(* Logix 5000 project; controller BTS01 vendor 1 type 14 code 217 rev 32.14; software revision 32.04; part 9 of 15 *)
(* tags used below, declared in another part *)
   Alarm_Active : DINT;
   Alarm_TMR : TIMER[17,32];
   ALM_ENABLE : DINT[25];
   HMI_Global_Alarm_Ack_PB : BOOL;
   HMIAlarms : DINT[25];   // Alarm Trigger Array
   HMIAlarmsMsg : STRING64[17,32];   // Alarm Descriptions to Match Alarm Trigger Array
(* Alarm, continued *)

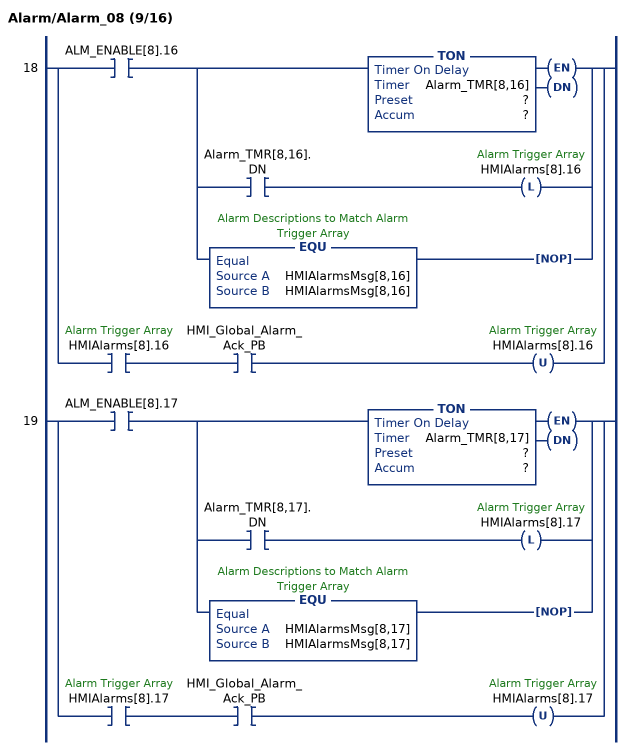
   [picture p159: Alarm/Alarm_08 rungs 18-19]
   18: [XIC(ALM_ENABLE[8].16) [TON(Alarm_TMR[8,16],?,?) ,XIC(Alarm_TMR[8,16].DN) OTL(HMIAlarms[8].16) ,EQU(HMIAlarmsMsg[8,16],HMIAlarmsMsg[8,16]) NOP() ] ,XIC(HMIAlarms[8].16) XIC(HMI_Global_Alarm_Ack_PB) OTU(HMIAlarms[8].16) ];
   19: [XIC(ALM_ENABLE[8].17) [TON(Alarm_TMR[8,17],?,?) ,XIC(Alarm_TMR[8,17].DN) OTL(HMIAlarms[8].17) ,EQU(HMIAlarmsMsg[8,17],HMIAlarmsMsg[8,17]) NOP() ] ,XIC(HMIAlarms[8].17) XIC(HMI_Global_Alarm_Ack_PB) OTU(HMIAlarms[8].17) ];
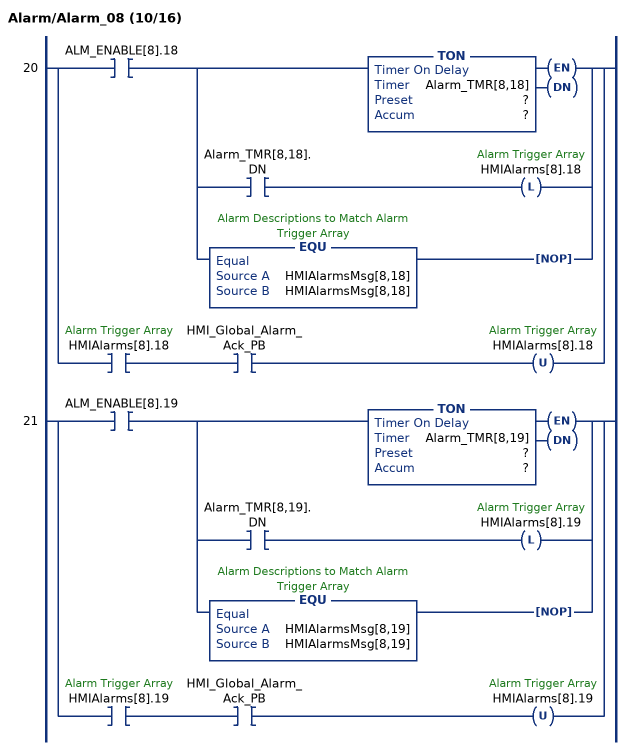
   20: [XIC(ALM_ENABLE[8].18) [TON(Alarm_TMR[8,18],?,?) ,XIC(Alarm_TMR[8,18].DN) OTL(HMIAlarms[8].18) ,EQU(HMIAlarmsMsg[8,18],HMIAlarmsMsg[8,18]) NOP() ] ,XIC(HMIAlarms[8].18) XIC(HMI_Global_Alarm_Ack_PB) OTU(HMIAlarms[8].18) ];
   21: [XIC(ALM_ENABLE[8].19) [TON(Alarm_TMR[8,19],?,?) ,XIC(Alarm_TMR[8,19].DN) OTL(HMIAlarms[8].19) ,EQU(HMIAlarmsMsg[8,19],HMIAlarmsMsg[8,19]) NOP() ] ,XIC(HMIAlarms[8].19) XIC(HMI_Global_Alarm_Ack_PB) OTU(HMIAlarms[8].19) ];
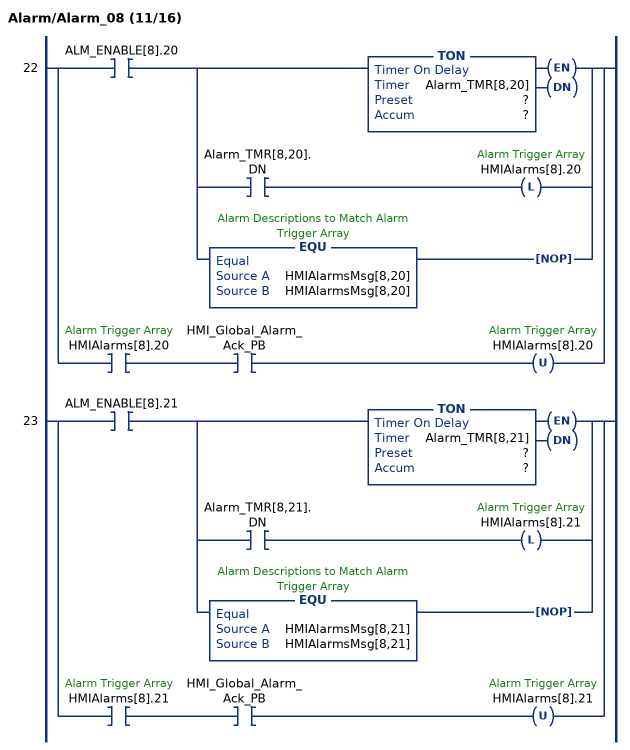
   22: [XIC(ALM_ENABLE[8].20) [TON(Alarm_TMR[8,20],?,?) ,XIC(Alarm_TMR[8,20].DN) OTL(HMIAlarms[8].20) ,EQU(HMIAlarmsMsg[8,20],HMIAlarmsMsg[8,20]) NOP() ] ,XIC(HMIAlarms[8].20) XIC(HMI_Global_Alarm_Ack_PB) OTU(HMIAlarms[8].20) ];
   23: [XIC(ALM_ENABLE[8].21) [TON(Alarm_TMR[8,21],?,?) ,XIC(Alarm_TMR[8,21].DN) OTL(HMIAlarms[8].21) ,EQU(HMIAlarmsMsg[8,21],HMIAlarmsMsg[8,21]) NOP() ] ,XIC(HMIAlarms[8].21) XIC(HMI_Global_Alarm_Ack_PB) OTU(HMIAlarms[8].21) ];
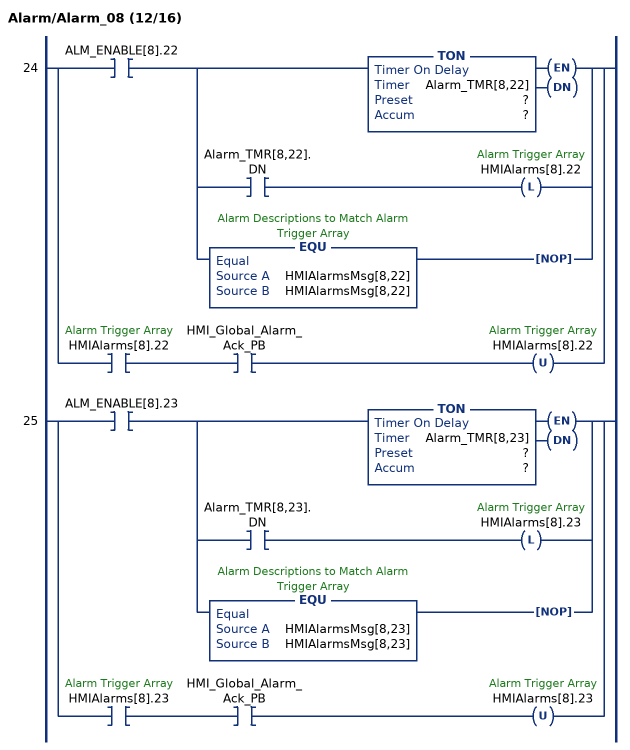
   24: [XIC(ALM_ENABLE[8].22) [TON(Alarm_TMR[8,22],?,?) ,XIC(Alarm_TMR[8,22].DN) OTL(HMIAlarms[8].22) ,EQU(HMIAlarmsMsg[8,22],HMIAlarmsMsg[8,22]) NOP() ] ,XIC(HMIAlarms[8].22) XIC(HMI_Global_Alarm_Ack_PB) OTU(HMIAlarms[8].22) ];
   25: [XIC(ALM_ENABLE[8].23) [TON(Alarm_TMR[8,23],?,?) ,XIC(Alarm_TMR[8,23].DN) OTL(HMIAlarms[8].23) ,EQU(HMIAlarmsMsg[8,23],HMIAlarmsMsg[8,23]) NOP() ] ,XIC(HMIAlarms[8].23) XIC(HMI_Global_Alarm_Ack_PB) OTU(HMIAlarms[8].23) ];
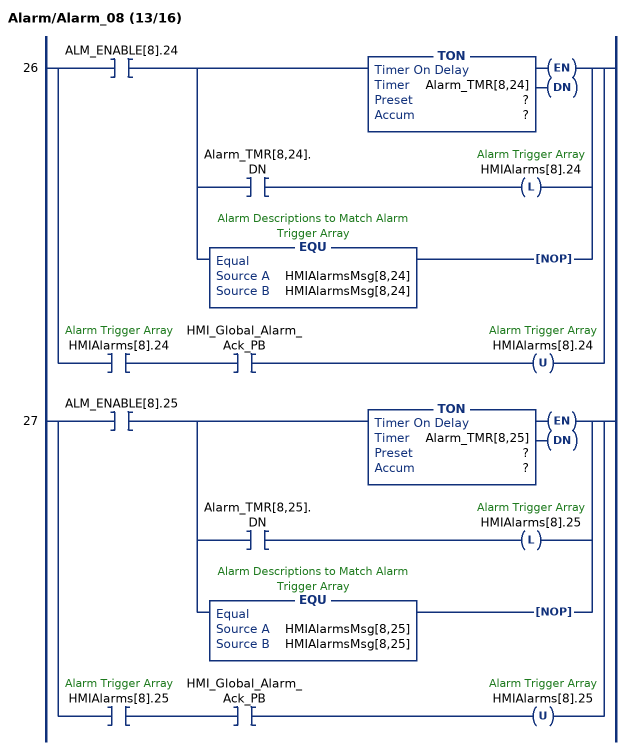
   26: [XIC(ALM_ENABLE[8].24) [TON(Alarm_TMR[8,24],?,?) ,XIC(Alarm_TMR[8,24].DN) OTL(HMIAlarms[8].24) ,EQU(HMIAlarmsMsg[8,24],HMIAlarmsMsg[8,24]) NOP() ] ,XIC(HMIAlarms[8].24) XIC(HMI_Global_Alarm_Ack_PB) OTU(HMIAlarms[8].24) ];
   27: [XIC(ALM_ENABLE[8].25) [TON(Alarm_TMR[8,25],?,?) ,XIC(Alarm_TMR[8,25].DN) OTL(HMIAlarms[8].25) ,EQU(HMIAlarmsMsg[8,25],HMIAlarmsMsg[8,25]) NOP() ] ,XIC(HMIAlarms[8].25) XIC(HMI_Global_Alarm_Ack_PB) OTU(HMIAlarms[8].25) ];
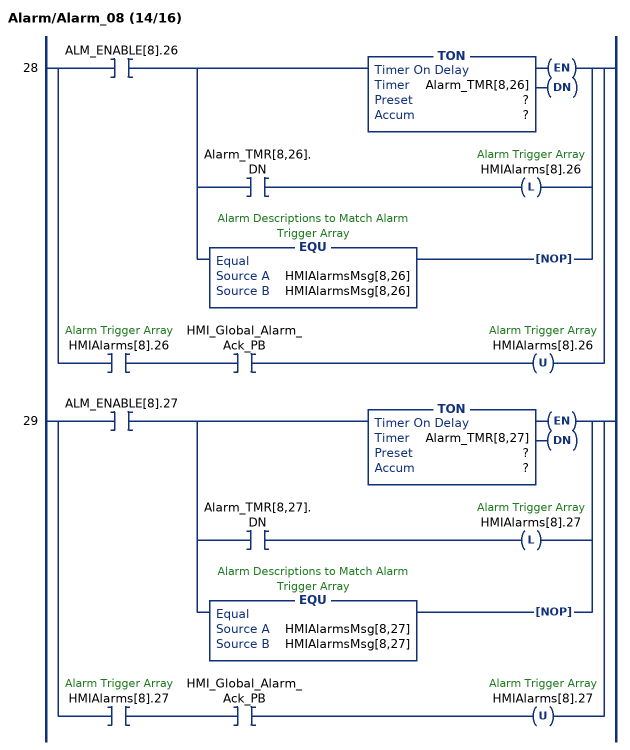
   28: [XIC(ALM_ENABLE[8].26) [TON(Alarm_TMR[8,26],?,?) ,XIC(Alarm_TMR[8,26].DN) OTL(HMIAlarms[8].26) ,EQU(HMIAlarmsMsg[8,26],HMIAlarmsMsg[8,26]) NOP() ] ,XIC(HMIAlarms[8].26) XIC(HMI_Global_Alarm_Ack_PB) OTU(HMIAlarms[8].26) ];
   29: [XIC(ALM_ENABLE[8].27) [TON(Alarm_TMR[8,27],?,?) ,XIC(Alarm_TMR[8,27].DN) OTL(HMIAlarms[8].27) ,EQU(HMIAlarmsMsg[8,27],HMIAlarmsMsg[8,27]) NOP() ] ,XIC(HMIAlarms[8].27) XIC(HMI_Global_Alarm_Ack_PB) OTU(HMIAlarms[8].27) ];
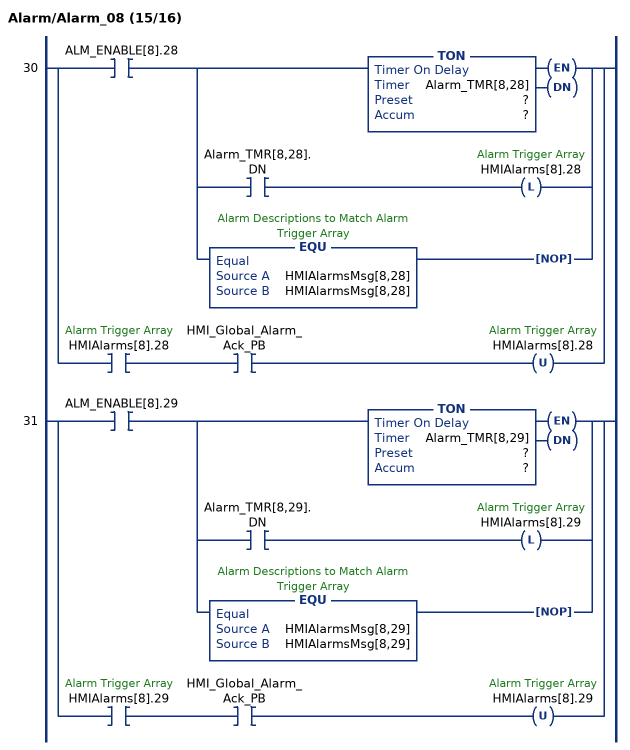
   30: [XIC(ALM_ENABLE[8].28) [TON(Alarm_TMR[8,28],?,?) ,XIC(Alarm_TMR[8,28].DN) OTL(HMIAlarms[8].28) ,EQU(HMIAlarmsMsg[8,28],HMIAlarmsMsg[8,28]) NOP() ] ,XIC(HMIAlarms[8].28) XIC(HMI_Global_Alarm_Ack_PB) OTU(HMIAlarms[8].28) ];
   31: [XIC(ALM_ENABLE[8].29) [TON(Alarm_TMR[8,29],?,?) ,XIC(Alarm_TMR[8,29].DN) OTL(HMIAlarms[8].29) ,EQU(HMIAlarmsMsg[8,29],HMIAlarmsMsg[8,29]) NOP() ] ,XIC(HMIAlarms[8].29) XIC(HMI_Global_Alarm_Ack_PB) OTU(HMIAlarms[8].29) ];
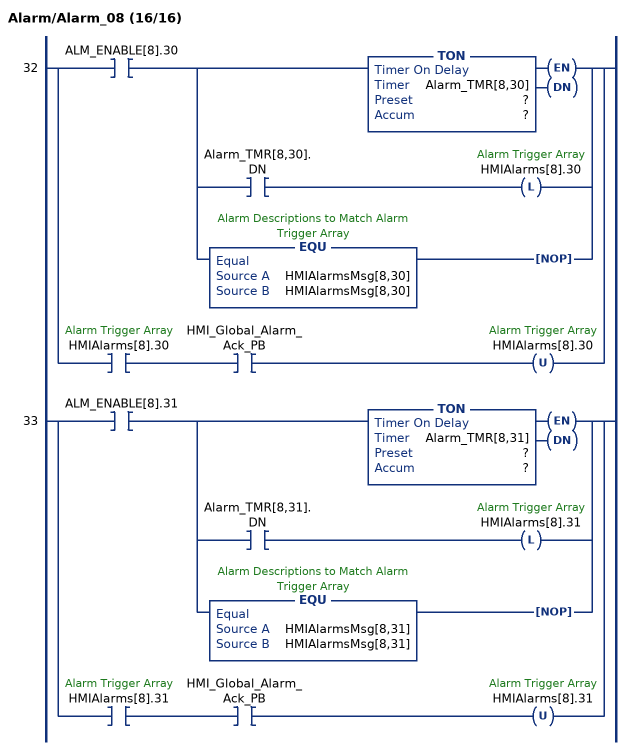
   32: [XIC(ALM_ENABLE[8].30) [TON(Alarm_TMR[8,30],?,?) ,XIC(Alarm_TMR[8,30].DN) OTL(HMIAlarms[8].30) ,EQU(HMIAlarmsMsg[8,30],HMIAlarmsMsg[8,30]) NOP() ] ,XIC(HMIAlarms[8].30) XIC(HMI_Global_Alarm_Ack_PB) OTU(HMIAlarms[8].30) ];
   33: [XIC(ALM_ENABLE[8].31) [TON(Alarm_TMR[8,31],?,?) ,XIC(Alarm_TMR[8,31].DN) OTL(HMIAlarms[8].31) ,EQU(HMIAlarmsMsg[8,31],HMIAlarmsMsg[8,31]) NOP() ] ,XIC(HMIAlarms[8].31) XIC(HMI_Global_Alarm_Ack_PB) OTU(HMIAlarms[8].31) ];
END_ROUTINE

ROUTINE Alarm_09   (* ladder *)
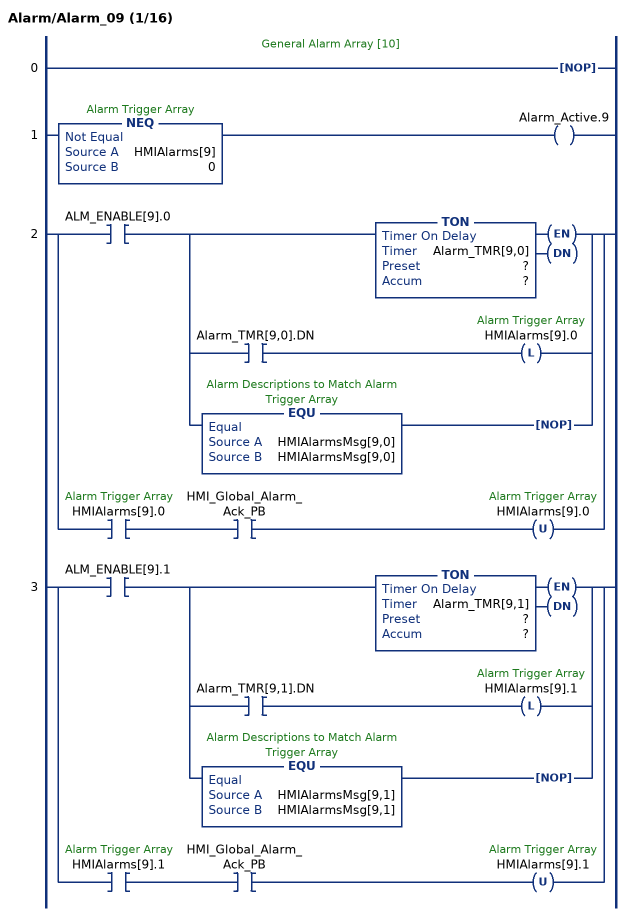
   // General Alarm Array [10]
   0: NOP();
   1: NEQ(HMIAlarms[9],0)OTE(Alarm_Active.9);
   2: [XIC(ALM_ENABLE[9].0) [TON(Alarm_TMR[9,0],?,?) ,XIC(Alarm_TMR[9,0].DN) OTL(HMIAlarms[9].0) ,EQU(HMIAlarmsMsg[9,0],HMIAlarmsMsg[9,0]) NOP() ] ,XIC(HMIAlarms[9].0) XIC(HMI_Global_Alarm_Ack_PB) OTU(HMIAlarms[9].0) ];
   3: [XIC(ALM_ENABLE[9].1) [TON(Alarm_TMR[9,1],?,?) ,XIC(Alarm_TMR[9,1].DN) OTL(HMIAlarms[9].1) ,EQU(HMIAlarmsMsg[9,1],HMIAlarmsMsg[9,1]) NOP() ] ,XIC(HMIAlarms[9].1) XIC(HMI_Global_Alarm_Ack_PB) OTU(HMIAlarms[9].1) ];
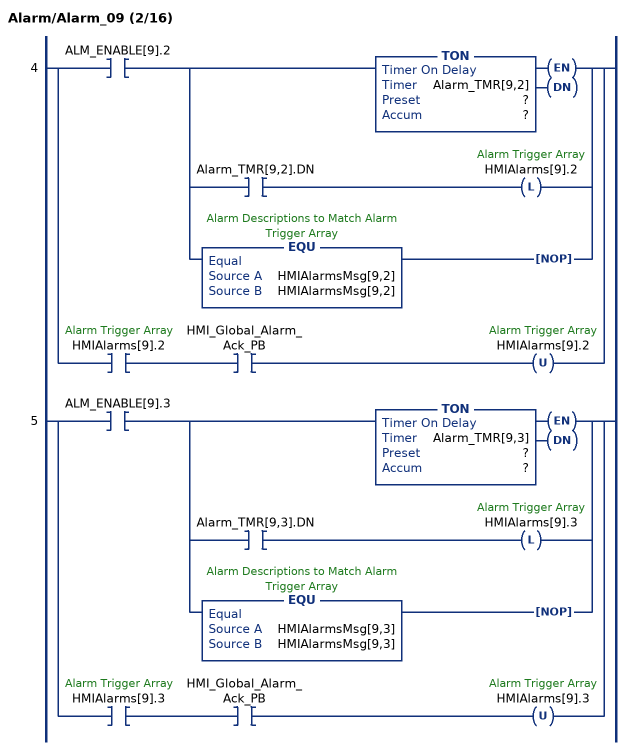
   4: [XIC(ALM_ENABLE[9].2) [TON(Alarm_TMR[9,2],?,?) ,XIC(Alarm_TMR[9,2].DN) OTL(HMIAlarms[9].2) ,EQU(HMIAlarmsMsg[9,2],HMIAlarmsMsg[9,2]) NOP() ] ,XIC(HMIAlarms[9].2) XIC(HMI_Global_Alarm_Ack_PB) OTU(HMIAlarms[9].2) ];
   5: [XIC(ALM_ENABLE[9].3) [TON(Alarm_TMR[9,3],?,?) ,XIC(Alarm_TMR[9,3].DN) OTL(HMIAlarms[9].3) ,EQU(HMIAlarmsMsg[9,3],HMIAlarmsMsg[9,3]) NOP() ] ,XIC(HMIAlarms[9].3) XIC(HMI_Global_Alarm_Ack_PB) OTU(HMIAlarms[9].3) ];
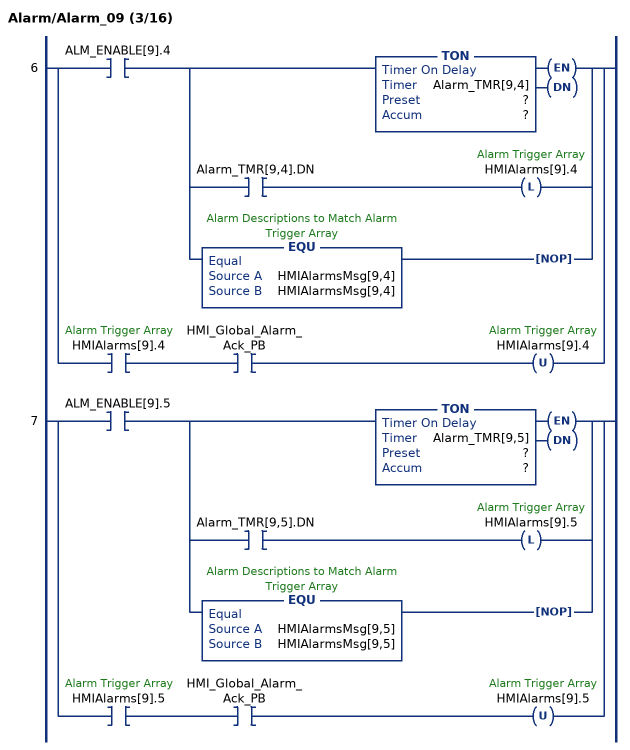
   6: [XIC(ALM_ENABLE[9].4) [TON(Alarm_TMR[9,4],?,?) ,XIC(Alarm_TMR[9,4].DN) OTL(HMIAlarms[9].4) ,EQU(HMIAlarmsMsg[9,4],HMIAlarmsMsg[9,4]) NOP() ] ,XIC(HMIAlarms[9].4) XIC(HMI_Global_Alarm_Ack_PB) OTU(HMIAlarms[9].4) ];
   7: [XIC(ALM_ENABLE[9].5) [TON(Alarm_TMR[9,5],?,?) ,XIC(Alarm_TMR[9,5].DN) OTL(HMIAlarms[9].5) ,EQU(HMIAlarmsMsg[9,5],HMIAlarmsMsg[9,5]) NOP() ] ,XIC(HMIAlarms[9].5) XIC(HMI_Global_Alarm_Ack_PB) OTU(HMIAlarms[9].5) ];
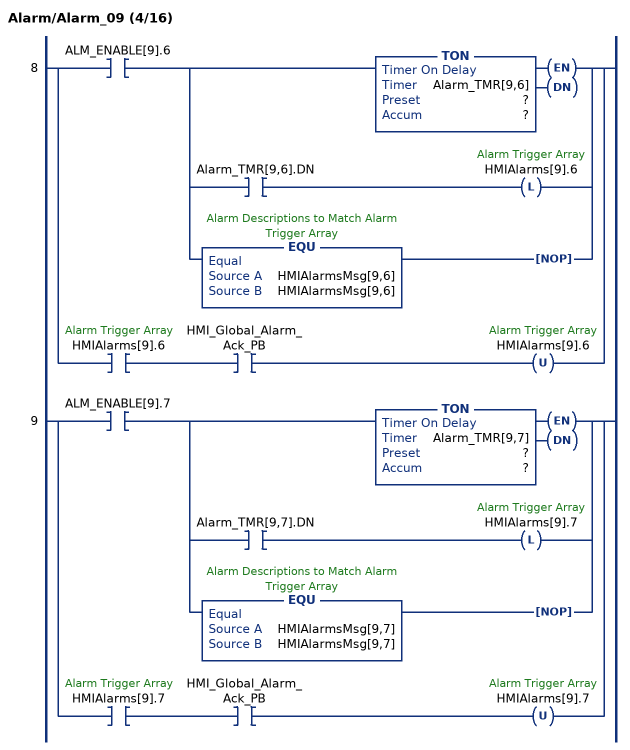
   8: [XIC(ALM_ENABLE[9].6) [TON(Alarm_TMR[9,6],?,?) ,XIC(Alarm_TMR[9,6].DN) OTL(HMIAlarms[9].6) ,EQU(HMIAlarmsMsg[9,6],HMIAlarmsMsg[9,6]) NOP() ] ,XIC(HMIAlarms[9].6) XIC(HMI_Global_Alarm_Ack_PB) OTU(HMIAlarms[9].6) ];
   9: [XIC(ALM_ENABLE[9].7) [TON(Alarm_TMR[9,7],?,?) ,XIC(Alarm_TMR[9,7].DN) OTL(HMIAlarms[9].7) ,EQU(HMIAlarmsMsg[9,7],HMIAlarmsMsg[9,7]) NOP() ] ,XIC(HMIAlarms[9].7) XIC(HMI_Global_Alarm_Ack_PB) OTU(HMIAlarms[9].7) ];
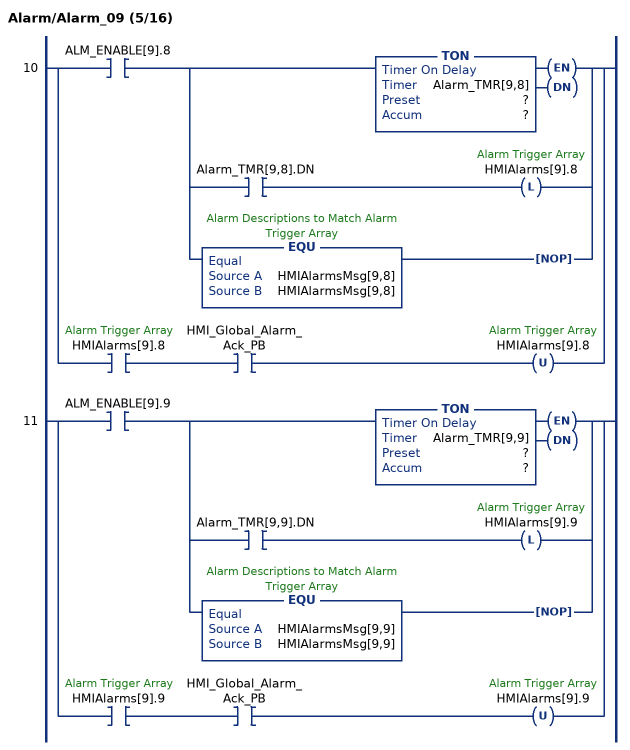
   10: [XIC(ALM_ENABLE[9].8) [TON(Alarm_TMR[9,8],?,?) ,XIC(Alarm_TMR[9,8].DN) OTL(HMIAlarms[9].8) ,EQU(HMIAlarmsMsg[9,8],HMIAlarmsMsg[9,8]) NOP() ] ,XIC(HMIAlarms[9].8) XIC(HMI_Global_Alarm_Ack_PB) OTU(HMIAlarms[9].8) ];
   11: [XIC(ALM_ENABLE[9].9) [TON(Alarm_TMR[9,9],?,?) ,XIC(Alarm_TMR[9,9].DN) OTL(HMIAlarms[9].9) ,EQU(HMIAlarmsMsg[9,9],HMIAlarmsMsg[9,9]) NOP() ] ,XIC(HMIAlarms[9].9) XIC(HMI_Global_Alarm_Ack_PB) OTU(HMIAlarms[9].9) ];
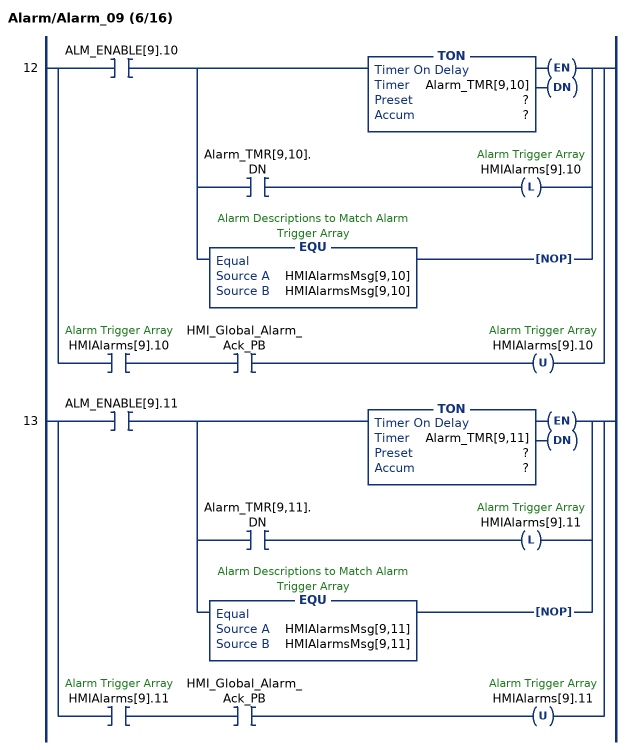
   12: [XIC(ALM_ENABLE[9].10) [TON(Alarm_TMR[9,10],?,?) ,XIC(Alarm_TMR[9,10].DN) OTL(HMIAlarms[9].10) ,EQU(HMIAlarmsMsg[9,10],HMIAlarmsMsg[9,10]) NOP() ] ,XIC(HMIAlarms[9].10) XIC(HMI_Global_Alarm_Ack_PB) OTU(HMIAlarms[9].10) ];
   13: [XIC(ALM_ENABLE[9].11) [TON(Alarm_TMR[9,11],?,?) ,XIC(Alarm_TMR[9,11].DN) OTL(HMIAlarms[9].11) ,EQU(HMIAlarmsMsg[9,11],HMIAlarmsMsg[9,11]) NOP() ] ,XIC(HMIAlarms[9].11) XIC(HMI_Global_Alarm_Ack_PB) OTU(HMIAlarms[9].11) ];
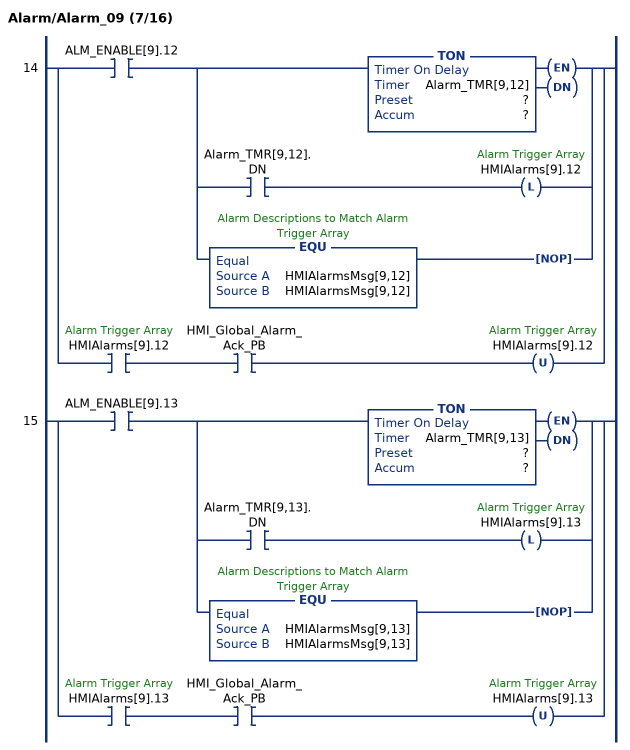
   14: [XIC(ALM_ENABLE[9].12) [TON(Alarm_TMR[9,12],?,?) ,XIC(Alarm_TMR[9,12].DN) OTL(HMIAlarms[9].12) ,EQU(HMIAlarmsMsg[9,12],HMIAlarmsMsg[9,12]) NOP() ] ,XIC(HMIAlarms[9].12) XIC(HMI_Global_Alarm_Ack_PB) OTU(HMIAlarms[9].12) ];
   15: [XIC(ALM_ENABLE[9].13) [TON(Alarm_TMR[9,13],?,?) ,XIC(Alarm_TMR[9,13].DN) OTL(HMIAlarms[9].13) ,EQU(HMIAlarmsMsg[9,13],HMIAlarmsMsg[9,13]) NOP() ] ,XIC(HMIAlarms[9].13) XIC(HMI_Global_Alarm_Ack_PB) OTU(HMIAlarms[9].13) ];
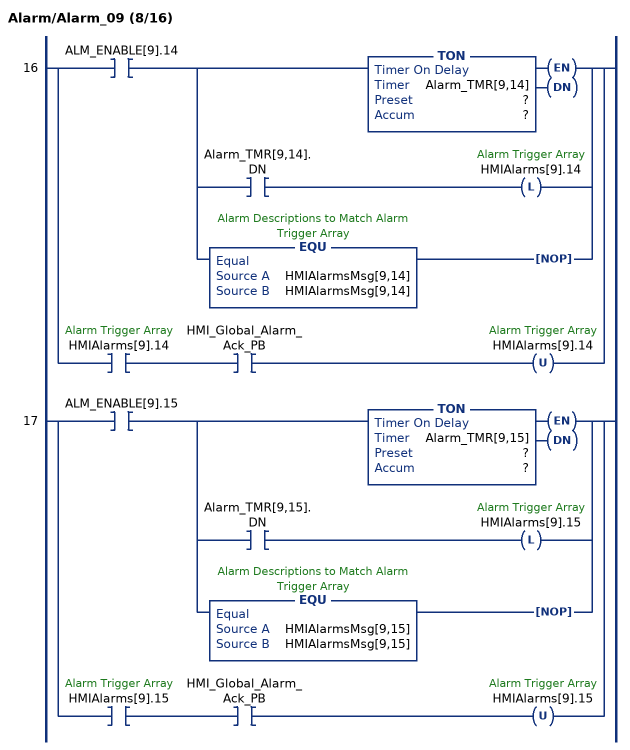
   16: [XIC(ALM_ENABLE[9].14) [TON(Alarm_TMR[9,14],?,?) ,XIC(Alarm_TMR[9,14].DN) OTL(HMIAlarms[9].14) ,EQU(HMIAlarmsMsg[9,14],HMIAlarmsMsg[9,14]) NOP() ] ,XIC(HMIAlarms[9].14) XIC(HMI_Global_Alarm_Ack_PB) OTU(HMIAlarms[9].14) ];
   17: [XIC(ALM_ENABLE[9].15) [TON(Alarm_TMR[9,15],?,?) ,XIC(Alarm_TMR[9,15].DN) OTL(HMIAlarms[9].15) ,EQU(HMIAlarmsMsg[9,15],HMIAlarmsMsg[9,15]) NOP() ] ,XIC(HMIAlarms[9].15) XIC(HMI_Global_Alarm_Ack_PB) OTU(HMIAlarms[9].15) ];
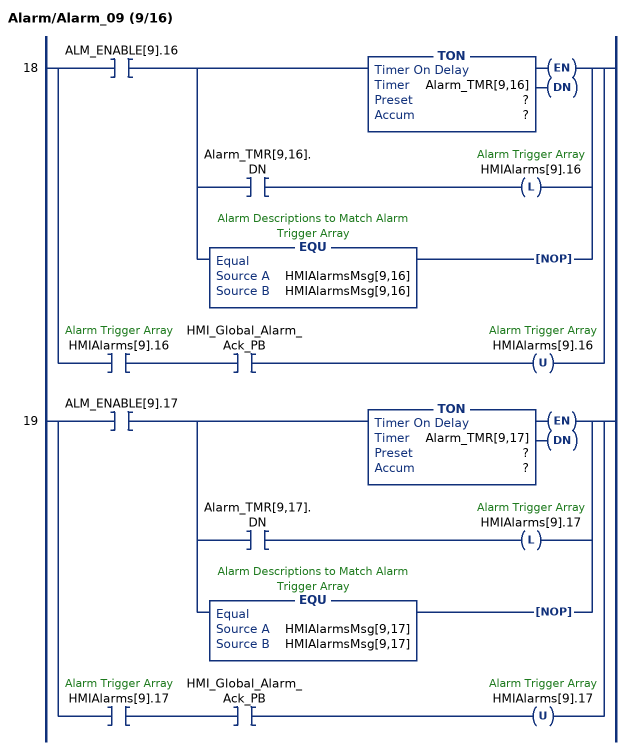
   18: [XIC(ALM_ENABLE[9].16) [TON(Alarm_TMR[9,16],?,?) ,XIC(Alarm_TMR[9,16].DN) OTL(HMIAlarms[9].16) ,EQU(HMIAlarmsMsg[9,16],HMIAlarmsMsg[9,16]) NOP() ] ,XIC(HMIAlarms[9].16) XIC(HMI_Global_Alarm_Ack_PB) OTU(HMIAlarms[9].16) ];
   19: [XIC(ALM_ENABLE[9].17) [TON(Alarm_TMR[9,17],?,?) ,XIC(Alarm_TMR[9,17].DN) OTL(HMIAlarms[9].17) ,EQU(HMIAlarmsMsg[9,17],HMIAlarmsMsg[9,17]) NOP() ] ,XIC(HMIAlarms[9].17) XIC(HMI_Global_Alarm_Ack_PB) OTU(HMIAlarms[9].17) ];
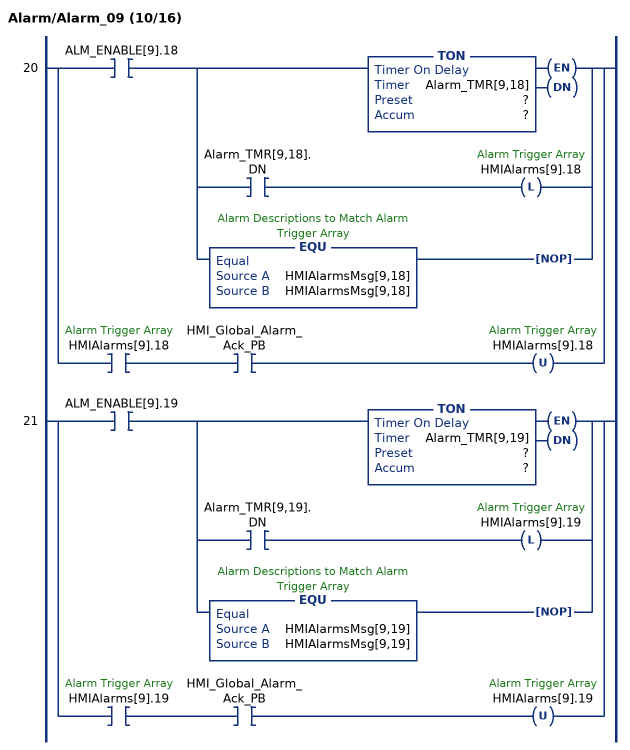
   20: [XIC(ALM_ENABLE[9].18) [TON(Alarm_TMR[9,18],?,?) ,XIC(Alarm_TMR[9,18].DN) OTL(HMIAlarms[9].18) ,EQU(HMIAlarmsMsg[9,18],HMIAlarmsMsg[9,18]) NOP() ] ,XIC(HMIAlarms[9].18) XIC(HMI_Global_Alarm_Ack_PB) OTU(HMIAlarms[9].18) ];
   21: [XIC(ALM_ENABLE[9].19) [TON(Alarm_TMR[9,19],?,?) ,XIC(Alarm_TMR[9,19].DN) OTL(HMIAlarms[9].19) ,EQU(HMIAlarmsMsg[9,19],HMIAlarmsMsg[9,19]) NOP() ] ,XIC(HMIAlarms[9].19) XIC(HMI_Global_Alarm_Ack_PB) OTU(HMIAlarms[9].19) ];
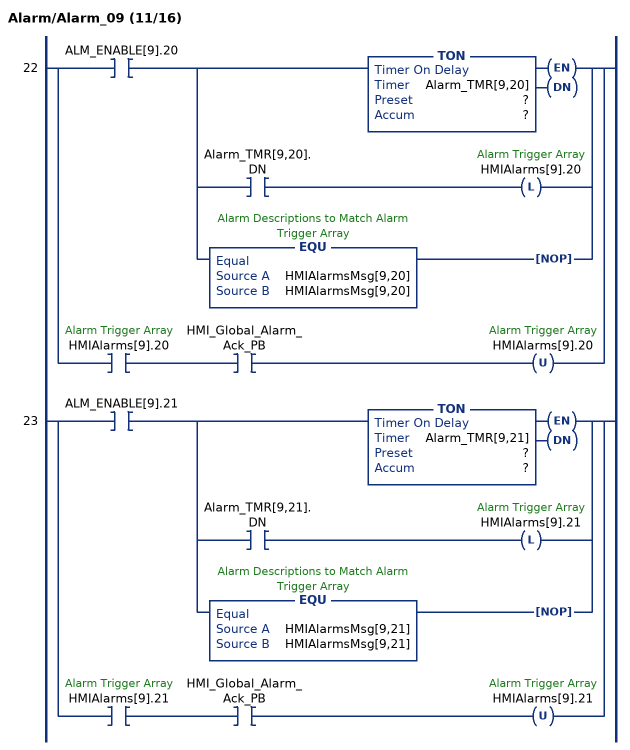
   22: [XIC(ALM_ENABLE[9].20) [TON(Alarm_TMR[9,20],?,?) ,XIC(Alarm_TMR[9,20].DN) OTL(HMIAlarms[9].20) ,EQU(HMIAlarmsMsg[9,20],HMIAlarmsMsg[9,20]) NOP() ] ,XIC(HMIAlarms[9].20) XIC(HMI_Global_Alarm_Ack_PB) OTU(HMIAlarms[9].20) ];
   23: [XIC(ALM_ENABLE[9].21) [TON(Alarm_TMR[9,21],?,?) ,XIC(Alarm_TMR[9,21].DN) OTL(HMIAlarms[9].21) ,EQU(HMIAlarmsMsg[9,21],HMIAlarmsMsg[9,21]) NOP() ] ,XIC(HMIAlarms[9].21) XIC(HMI_Global_Alarm_Ack_PB) OTU(HMIAlarms[9].21) ];
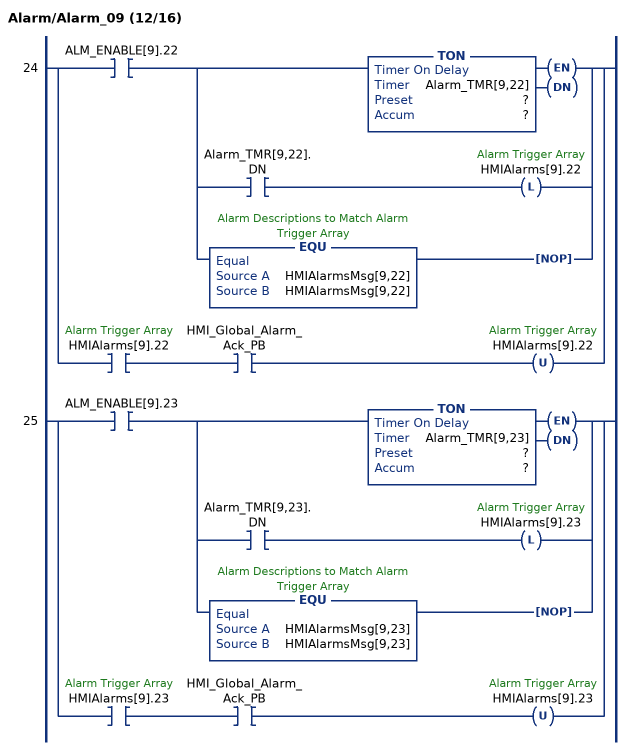
   24: [XIC(ALM_ENABLE[9].22) [TON(Alarm_TMR[9,22],?,?) ,XIC(Alarm_TMR[9,22].DN) OTL(HMIAlarms[9].22) ,EQU(HMIAlarmsMsg[9,22],HMIAlarmsMsg[9,22]) NOP() ] ,XIC(HMIAlarms[9].22) XIC(HMI_Global_Alarm_Ack_PB) OTU(HMIAlarms[9].22) ];
   25: [XIC(ALM_ENABLE[9].23) [TON(Alarm_TMR[9,23],?,?) ,XIC(Alarm_TMR[9,23].DN) OTL(HMIAlarms[9].23) ,EQU(HMIAlarmsMsg[9,23],HMIAlarmsMsg[9,23]) NOP() ] ,XIC(HMIAlarms[9].23) XIC(HMI_Global_Alarm_Ack_PB) OTU(HMIAlarms[9].23) ];
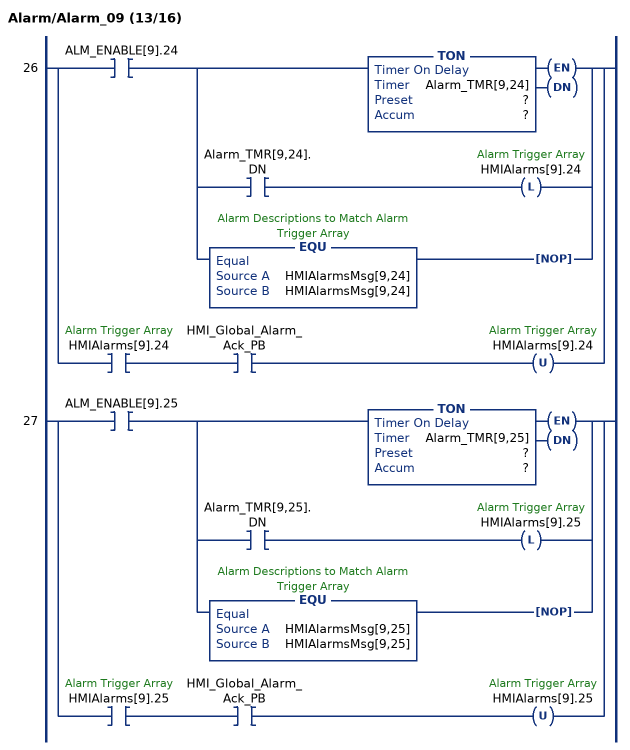
   26: [XIC(ALM_ENABLE[9].24) [TON(Alarm_TMR[9,24],?,?) ,XIC(Alarm_TMR[9,24].DN) OTL(HMIAlarms[9].24) ,EQU(HMIAlarmsMsg[9,24],HMIAlarmsMsg[9,24]) NOP() ] ,XIC(HMIAlarms[9].24) XIC(HMI_Global_Alarm_Ack_PB) OTU(HMIAlarms[9].24) ];
   27: [XIC(ALM_ENABLE[9].25) [TON(Alarm_TMR[9,25],?,?) ,XIC(Alarm_TMR[9,25].DN) OTL(HMIAlarms[9].25) ,EQU(HMIAlarmsMsg[9,25],HMIAlarmsMsg[9,25]) NOP() ] ,XIC(HMIAlarms[9].25) XIC(HMI_Global_Alarm_Ack_PB) OTU(HMIAlarms[9].25) ];
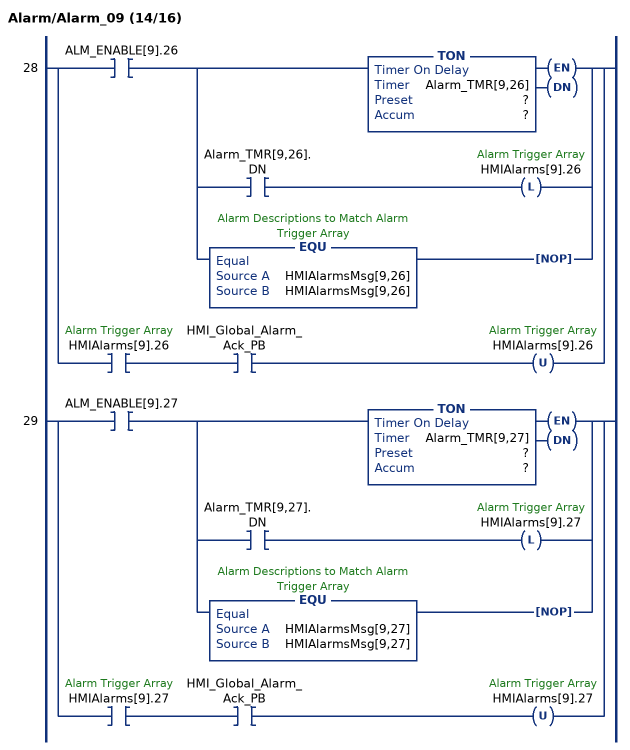
   28: [XIC(ALM_ENABLE[9].26) [TON(Alarm_TMR[9,26],?,?) ,XIC(Alarm_TMR[9,26].DN) OTL(HMIAlarms[9].26) ,EQU(HMIAlarmsMsg[9,26],HMIAlarmsMsg[9,26]) NOP() ] ,XIC(HMIAlarms[9].26) XIC(HMI_Global_Alarm_Ack_PB) OTU(HMIAlarms[9].26) ];
   29: [XIC(ALM_ENABLE[9].27) [TON(Alarm_TMR[9,27],?,?) ,XIC(Alarm_TMR[9,27].DN) OTL(HMIAlarms[9].27) ,EQU(HMIAlarmsMsg[9,27],HMIAlarmsMsg[9,27]) NOP() ] ,XIC(HMIAlarms[9].27) XIC(HMI_Global_Alarm_Ack_PB) OTU(HMIAlarms[9].27) ];
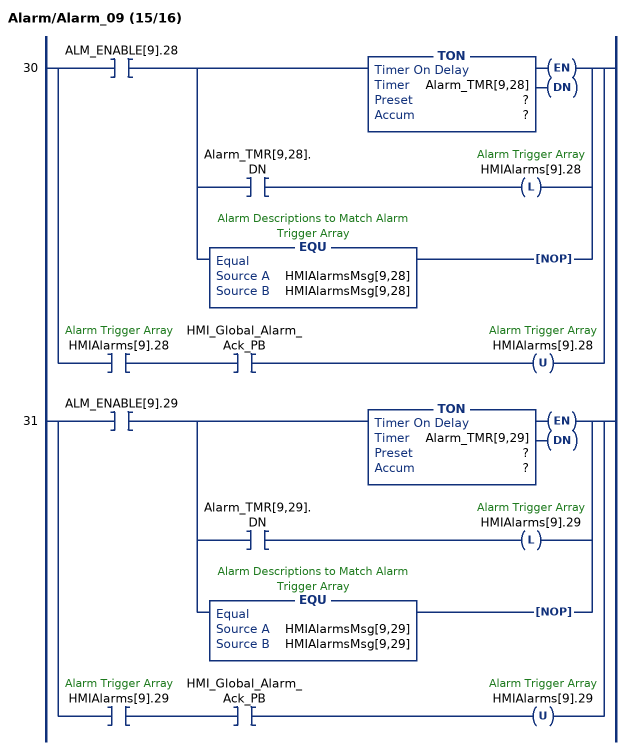
   30: [XIC(ALM_ENABLE[9].28) [TON(Alarm_TMR[9,28],?,?) ,XIC(Alarm_TMR[9,28].DN) OTL(HMIAlarms[9].28) ,EQU(HMIAlarmsMsg[9,28],HMIAlarmsMsg[9,28]) NOP() ] ,XIC(HMIAlarms[9].28) XIC(HMI_Global_Alarm_Ack_PB) OTU(HMIAlarms[9].28) ];
   31: [XIC(ALM_ENABLE[9].29) [TON(Alarm_TMR[9,29],?,?) ,XIC(Alarm_TMR[9,29].DN) OTL(HMIAlarms[9].29) ,EQU(HMIAlarmsMsg[9,29],HMIAlarmsMsg[9,29]) NOP() ] ,XIC(HMIAlarms[9].29) XIC(HMI_Global_Alarm_Ack_PB) OTU(HMIAlarms[9].29) ];
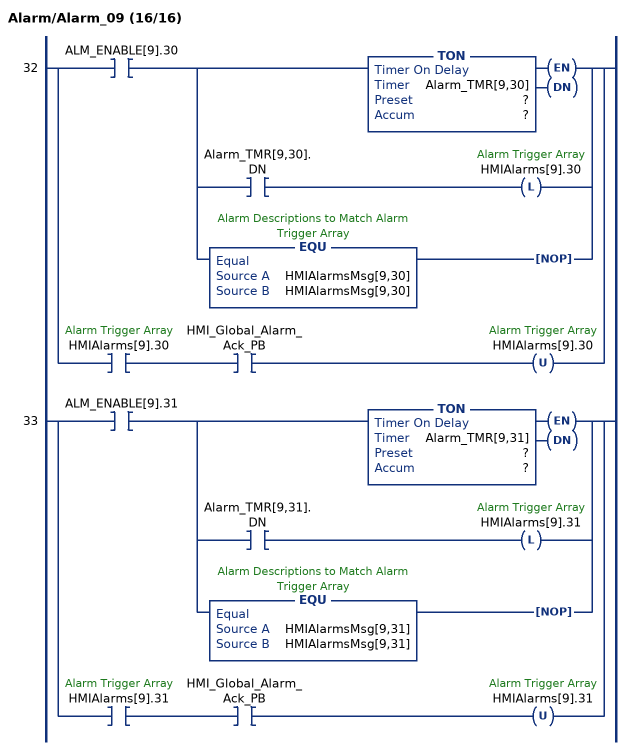
   32: [XIC(ALM_ENABLE[9].30) [TON(Alarm_TMR[9,30],?,?) ,XIC(Alarm_TMR[9,30].DN) OTL(HMIAlarms[9].30) ,EQU(HMIAlarmsMsg[9,30],HMIAlarmsMsg[9,30]) NOP() ] ,XIC(HMIAlarms[9].30) XIC(HMI_Global_Alarm_Ack_PB) OTU(HMIAlarms[9].30) ];
   33: [XIC(ALM_ENABLE[9].31) [TON(Alarm_TMR[9,31],?,?) ,XIC(Alarm_TMR[9,31].DN) OTL(HMIAlarms[9].31) ,EQU(HMIAlarmsMsg[9,31],HMIAlarmsMsg[9,31]) NOP() ] ,XIC(HMIAlarms[9].31) XIC(HMI_Global_Alarm_Ack_PB) OTU(HMIAlarms[9].31) ];
END_ROUTINE
